// TIA Portal V20 export
TYPE "ASI_GW_DATOS"
   STRUCT
      nameOfStation : String;
      ipAdress : Array[0..3] of USInt;
   END_STRUCT;
END_TYPE
